(*
SPDX-FileCopyrightText: © 2026 Oleksandr Tiutyk <trofimich@gmail.com>
SPDX-License-Identifier: MIT
License: https://opensource.org/license/mit
*)

INTERFACE IInvalidWorkflowTransitionException EXTENDS TOF_Core.IGeneralException

METHOD Throw
VAR_INPUT
	sourceNamespaceName : STRING;
	sourceClassName : STRING;
	sourcePOUName : STRING;
	sourcePosition : STRING;
	fromState : WORKFLOW_ELEMENT_STATE;
	toState : WORKFLOW_ELEMENT_STATE;
END_VAR
END_METHOD

END_INTERFACE

(* stored: Version 1.1.0.1
   Itf IInvalidWorkflowTransitionException: Id {7340e873-0fee-42d6-bda3-e9bfd586f0f4}
   Method Throw: Id {6c679139-20ab-4061-b94a-4c6f3303172c} *)
